{attribute 'GeneratedUsingTerminal: ER8309-1022-0018'}
{attribute addProperty BoxType "ER8309-1022-0018"}
{attribute addProperty Id "StatusAT %I*Status_6CCA259F6Rotational_SpeedAT %I*INT2Rotation_DirectionAT %I*UINT2"}
{attribute addProperty CRC "3274820158"}
{attribute addProperty Size "10"}
TYPE TACHO_Single_Shaft_Mode_Input_Channel_C331CA3E EXTENDS InputBase_8311D824 :
STRUCT
	{attribute addProperty Name "Status"}
	Status AT %I* : Status_6CCA259F;
	{attribute addProperty Name "Rotational_Speed"}
	Rotational_Speed AT %I* : INT;
	{attribute addProperty Name "Rotation_Direction"}
	Rotation_Direction AT %I* : UINT;
END_STRUCT
END_TYPE

(* stored: Version 1.2.0.0, ProductVersion 3.1.4024.11
   DUT TACHO_Single_Shaft_Mode_Input_Channel_C331CA3E: Id {4d4c4678-fbad-43d9-85f2-f92f57127ff4} *)
